FUNCTION_BLOCK FB_MotionRef_1
VAR_INPUT
	
END_VAR
VAR_OUTPUT
	
END_VAR
VAR
	
END_VAR

END_FUNCTION_BLOCK

(* stored: Version 1.1.0.1
   POU FB_MotionRef_1: Id {f1bb715d-1607-45e3-9371-643846e54291}, SpecialFunc None *)
